ABB RobotStudio station: ABBPracticalTraining_1.rsstnx

Station ABBPracticalTraining (saved by RobotStudio 25.2.11220.0)
Controller IRB2600_12_165
  mechanical unit ROB_1: IRB2600_12_165__02, 6 joints, base frame (0, 0, 0) mm
Layout (positions relative to the parent item):
  - IRB2600_12_165__02 [mechanism, from %ABB.RobotStudio.Models.IRB2600%\IRB2600_12_165_G_02.rslib] at (0, 0, 0) mm; joint values [1.1412, -0.813, 0.8329, 3.1517, -0.4917, -3.1683] (rad or m)
  - MyTool [mechanism, from Training Objects\myTool.rslib] at (213.2, 466.4, 983.63) mm, rotated rx -178.45 ry 60.67 rz -112.52 deg
  - table_and_fixture_140 [part] at (363.72, 396.2, 0) mm, size 450 x 350 x 308 mm
  - Curve_thing [part, from Training Objects\Curve_Thing.rslib] at (388.72, 421.21, 308) mm
Attachment: MyTool is attached to IRB2600_12_165__02 / Link6
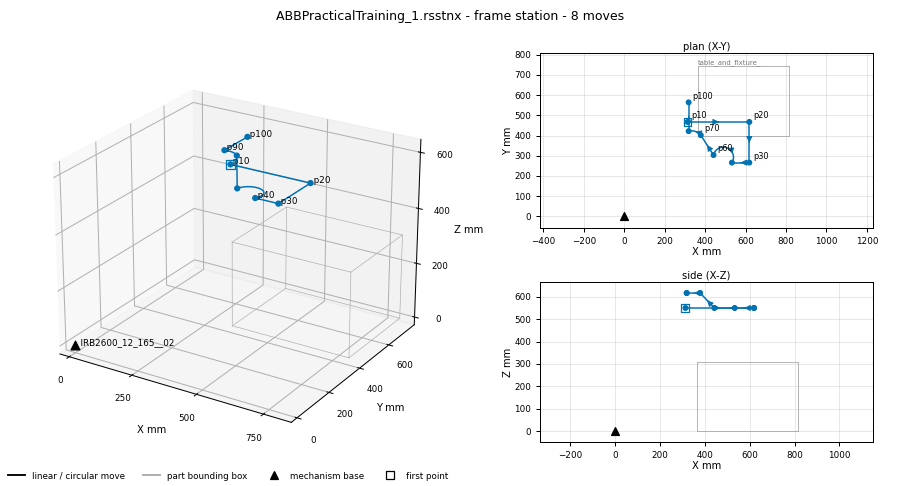
[picture p0: tool path of ABBPracticalTraining_1.rsstnx in frame station, 8 of 10 moves have a stored position in this frame; points joined in program order, loops and branches not executed]
Targets, tools, work objects and paths stored in the station, written as RAPID:
! task T_ROB1
MODULE CalibData
  PERS tooldata MyTool:=[TRUE,[[31.792631019,0,229.638935148],[0.945518576,0,0.325568154,0]],[1,[0,0,1],[1,0,0,0],0,0,0]];
  TASK PERS wobjdata Workobject_1:=[FALSE,TRUE,"",[[788.717,721.202,308],[0,0,0,1]],[[0,0,0],[1,0,0,0]]];
ENDMODULE

! task T_ROB1
MODULE Module1
  CONST jointtarget jpos10:=[[65.3885,-46.5801,47.724,180.577,-28.1733,-181.532],[9E+09,9E+09,9E+09,9E+09,9E+09,9E+09]];
  CONST robtarget p10:=[[312.95,467.14,549.66],[0.426451,-0.473639,0.72144,0.270795],[0,3,-4,1],[9E+09,9E+09,9E+09,9E+09,9E+09,9E+09]];
  CONST robtarget p20:=[[618.74,467.14,549.66],[0.42645,-0.473638,0.721441,0.270796],[0,3,-4,1],[9E+09,9E+09,9E+09,9E+09,9E+09,9E+09]];
  CONST robtarget p30:=[[618.74,265.86,549.66],[0.42645,-0.473638,0.721441,0.270796],[0,3,-4,1],[9E+09,9E+09,9E+09,9E+09,9E+09,9E+09]];
  CONST robtarget p40:=[[532.78,265.86,549.66],[0.42645,-0.473638,0.721441,0.270796],[0,3,-4,1],[9E+09,9E+09,9E+09,9E+09,9E+09,9E+09]];
  CONST robtarget p50:=[[527,326.42,549.66],[0.42645,-0.473638,0.721441,0.270795],[0,3,-4,1],[9E+09,9E+09,9E+09,9E+09,9E+09,9E+09]];
  CONST robtarget p60:=[[441.64,303.39,549.66],[0.42645,-0.473639,0.721441,0.270795],[0,3,-4,1],[9E+09,9E+09,9E+09,9E+09,9E+09,9E+09]];
  CONST robtarget p70:=[[378.59,401.65,616.69],[0.282515,-0.571295,0.767786,0.0656612],[0,2,-3,1],[9E+09,9E+09,9E+09,9E+09,9E+09,9E+09]];
  CONST robtarget p80:=[[352.21,419.85,616.31],[0.282515,-0.571296,0.767786,0.0656606],[0,1,-3,1],[9E+09,9E+09,9E+09,9E+09,9E+09,9E+09]];
  CONST robtarget p90:=[[318.51,421.57,616.31],[0.282515,-0.571296,0.767786,0.0656604],[0,1,-3,1],[9E+09,9E+09,9E+09,9E+09,9E+09,9E+09]];
  CONST robtarget p100:=[[318.51,564.09,616.31],[0.282515,-0.571296,0.767786,0.0656605],[0,1,-2,1],[9E+09,9E+09,9E+09,9E+09,9E+09,9E+09]];
  PROC main()
    MoveAbsJ jpos10\NoEOffs,v1000,z50,tool0;
    MoveJ p10,v1000,fine,tool0;
    MoveL p20,v1000,fine,tool0;
    MoveL p30,v1000,fine,tool0;
    MoveL p40,v1000,fine,tool0;
    MoveC p50,p60,v1000,fine,tool0;
    MoveL p70,v1000,fine,tool0;
    MoveC p80,p90,v1000,fine,tool0;
    MoveL p100,v1000,fine,tool0;
    MoveAbsJ jpos10\NoEOffs,v1000,fine,tool0;
  ENDPROC
ENDMODULE

